Staubli VAL3: isListEmpty.pgx

public program isListEmpty(bool& x_bEmpty[])
begin
  if size(sItems)==1 and sItems[0]==""
    x_bEmpty=true
  else
    x_bEmpty=false
  endIf
end
